// TIA Portal V19 export
DATA_BLOCK "PopUpBitToScada"   // DB36
{ S7_Optimized_Access := 'TRUE' }
AUTHOR : FLA
FAMILY : UHT
VERSION : 1.0
// stored: AutoNumber false, MemoryReserve 0
   VAR RETAIN
      PC_number_from_intouch : Int;   // PC number from intouch - Range 1 to 8
      Count_down_to_reset : Int := -1;   // Count down to reset text number to pc x
      Pop_up_text_to_PC1 : Int;   // Pop up text number to intouch PC 1
      Pop_up_text_to_PC2 : Int;   // Pop up text number to intouch PC 2
      Pop_up_text_to_PC3 : Int;   // Pop up text number to intouch PC 3
      Pop_up_text_to_PC4 : Int;   // Pop up text number to intouch PC 4
      Pop_up_text_to_PC5 : Int;   // Pop up text number to intouch PC 5
      Pop_up_text_to_PC6 : Int;   // Pop up text number to intouch PC 6
      Pop_up_text_to_PC7 : Int;   // Pop up text number to intouch PC 7
      Pop_up_text_to_PC8 : Int;   // Pop up text number to intouch PC 8
      Pop_up_text_to_PC9 : Int;
      Monitor_comm_from_intouc : Int := -7535;   // Counter - Monitor comm. from intouch
   END_VAR
BEGIN
END_DATA_BLOCK
